Fanuc KAREL source: kt00939.KL

-- PROVISIONAL review KL for V940-1; original PC SHA256 b53cfca74661d560b3fb5231b164a15981249edd7cc302a32dbc98946a0a3f25
-- Incomplete behavior may be omitted. Consult companion uncertainty JSON. Do not deploy.
PROGRAM KT00939
%NOLOCKGROUP
VAR
  ENTRY : INTEGER
  PNAME : STRING[80]
  VNAME : STRING[80]
  STATUS : INTEGER
-- UNRESOLVED_DECL VALUE type=000101
BEGIN
  -- V9_ZERO_TABLE_METADATA_HINT layout=0001; no indexed target words; source/name/runtime held
  -- UNRESOLVED_PC offsets 5-12; opcodes 9C,23
  -- UNRESOLVED_PC offsets 17-25; opcodes 3F,75
  -- UNRESOLVED_PC offsets 30-43; opcodes 3F,75
  -- UNRESOLVED_PC offsets 48-92; opcodes 27,22,22,2A,22,2A,22,1C,22,AF
  -- UNRESOLVED_PC offsets 97-101; opcodes 7F
END KT00939
